_CFC_ (* Continuous Function Chart, elements in execution order *)
#0 MOVE(EN: NOT #25.Q1, SHU6_P2_M_MAXSPEED)
#1 SHU6_P2_SPEEDMOTOR <= #0
#2 OR(SHU6_P2_UST_RE_RABOTA, SHU6_P2_UST_RE_PUSK)
#3 AND(SHU6_P2_YA3_M_UST_VKL_UVEL_CHAST, SHU6_P2_TE6_TE_NM_UST)
#4 AND(SHU6_P2_YA4_M_UST_VKL_UVEL_CHAST, SHU6_P2_TE6_TE_NB_UST)
#5 AND(#3, #4)
#6 OR(SHU6_P2_TE6_TE_M_UST, SHU6_P2_TE6_TE_B_UST, SHU6_P2_UST_RE_STOP)
#7 AND(SHU6_P2_YA3_B_UST_VKL_STER_REG, SHU6_P2_TE6_TE_M_UST)
#8 AND(SHU6_P2_TE6_TE_B_UST, SHU6_P2_YA4_B_UST_VKL_STER_REG)
#9 OR(#7, #8)
#10 AND(SHU6_P2_OBRBSM, SHU6_P2_SA1_DO1)
#11 AND(#5, #10)
#12 SR_START_POV_REG:RS(SET: #11, RESET1: #6)
#13 AND(#9, #10)
#14 AND(#2, SHU6_P2_SA1_DO1)
#15 OR(SHU6_P2_UST_RE_RABOTA, #14)
#16 SEL(#12.Q1, SHU6_P2_SPEEDMOTOR, SHU6_P2_M_MAXSPEED)
#17 AND(SHU6_P2_YA4_M_UST_VKL_STER_REG, SHU6_P2_TE6_TE_B_UST)
#18 AND(#12.Q1, #14)
#19 SEL(#18, SHU6_P2_M_USKORENIE_PUSK, SHU6_P2_M_USKORENIE_UPR)
#20 AND(SHU6_P2_TE6_TE_NB_UST, SHU6_P2_YA4_M_UST_VKL_STER_REG)
#21 AND(SHU6_P2_YA3_M_UST_VKL_STER_REG, SHU6_P2_TE6_TE_NM_UST)
#22 SEL(SHU6_P2_UST_ZIMA, #20, #21)
#23 AND(#17, #22)
#24 OR(SHU6_P2_UST_RE_STOP, #23)
#25 SR_START_STER_REG:SR(SET1: #13, RESET: #24)
#26 AND(SHU6_P2_M_SB2_STER_REG, NOT #25.Q1)
#27 MOVE(EN: #26, SHU6_P2_M_MAXSPEED)
#28 SHU6_P2_SPEEDMOTOR <= #27
#29 OR(#12.Q1, #25.Q1)
#30 SEL(#25.Q1, #16, SHU6_P2_M_MINSPEED)
#31 SEL(#15, 0, #30)
#32 AND(#14, #25.Q1)
#33 SEL(#32, SHU6_P2_M_ZAMEDLENIE_OST, SHU6_P2_M_ZAMEDLENIE_UPR)
#34 SEL(SHU6_P2_UST_SET_STOP, #33, 1000)
#35 RR:RAMP_REAL(#31, #19, #34, T#1s, -)
#36 MOVE(EN: #29, #35)
#37 SHU6_P2_SPEEDMOTOR <= #36
#38 MOVE(EN: SHU6_P2_SA1_DO1, #35)
#39 SEL(#38.ENO, 0, #38)
#40 SEL(SHU6_P2_SA1_DI2_M, #39, SHU6_P2_M_ZAD_RUCH)
#41 SHU6_P2_ZAD_VN <= #40
#42 RT_KOMVKL_1:R_TRIG(CLK: SHU6_P2_UST_RE_PUSK)
#43 MOVE(EN: #42.Q, SHU6_P2_M_MAXSPEED)
#44 SHU6_P2_SPEEDMOTOR <= #43
#45 RT_KOMVKL_2:R_TRIG(CLK: TRUE)
#46 MOVE(EN: #45.Q, 5)
#47 SHU6_P2_M_ZAD_RUCH <= #46
#48 MOVE(EN: SHU6_V2_SA3_DO3, #35)
#49 SEL(#48.ENO, 0, #48)
#50 SEL(SHU6_V2_SA2_DI6_M, #49, SHU6_V2_M_ZAD_RUCH)
#51 SHU6_V2_ZAD_VN <= #50
_END_CFC_
END_PROGRAM
